PROGRAM RC4_CRYPT_DEMO_1
VAR
	RC4_CRYPT_STREAM: RC4_CRYPT_STREAM;
	(* buf : ARRAY [0..63] OF BYTE := 107,117,114,116;*) (* kurt *)
	buf : ARRAY [0..63] OF BYTE := 110,60,3,219; (* crypt *)
	mode: INT;
	key: STRING := '1234';
	size: UDINT := 4;
	pos: UDINT;
END_VAR

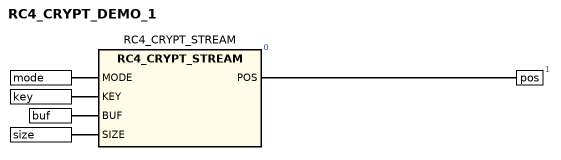
RC4_CRYPT_STREAM(MODE := mode, KEY := key, BUF := buf, SIZE := size);
pos := RC4_CRYPT_STREAM.POS;

END_PROGRAM

(* stored: Version 1.1.0.1, ProductVersion 3.1.4024.0
   POU RC4_CRYPT_DEMO_1: Id {b67aa629-a34e-4759-a216-6e2525b41127}, SpecialFunc None *)
